(* CODESYS project Proyecto_Mezclador_de_alimenos_Codesys_V3_5_Sp12 (1).export

Project tree, tasks and I/O mapping:
  Device : CPX-CEC-C1-V3, Festo AG & Co. KG, order no. 3473128, version 3.5.12.60
      unmapped channels: Rotary switch
    application Application
      libraries: Standard, * (System); Util, * (System)
      task MainTask (cyclic, interval t#250MS, priority 20) calls LUCES, MODOMANUAL, CriaTilapia, TilapiaJoven, Tilapiaenengorda, GRANOSANIM, FlechasANIM, FORMULAS_Y_LLENADO_DE_SILOS, Alertas_silo, Alertas_SiloX
      global variables GVL
      image pool ImagePool
      image pool ImagePool_1
      program Alertas_silo [ST]
      program Alertas_SiloX [LD]
      program CriaTilapia [LD]
      program FlechasANIM [LD]
      program FORMULAS_Y_LLENADO_DE_SILOS [LD]
      program GRANOSANIM [LD]
      program LUCES [ST]
      program MODOMANUAL [LD]
      program Tilapiaenengorda [LD]
      program TilapiaJoven [LD]
      Symbols
      text list TextList
      visualisation Visualization
    PLC_Diagnosis : PLC-Diagnosis, Festo AG & Co. KG, version 3.5.4.3
    CPX_System : CPX_System, Festo AG & Co. KG, order no. 3473128, version 1.278
*)

// Device/Application/GVL
VAR_GLOBAL
	
	ON: BOOL;
	OFF: BOOL;
	ResetS: BOOL;
	OPCIONES:INT;
	
	A1:REAL;
	A2:REAL;
	A3:REAL;
	
	VMotor1: REAL;
	VMotor2: REAL;
	VMotor3: REAL; 
	INICIO2: BOOL;
	
	SiloF: REAL;
	LSiloF: BOOL;
	
	APAGADO: BOOL;
	Apagado2: BOOL;
	
	LMotor1: BOOL;
	LMotor2: BOOL;
	LMotor3: BOOL;
	
	
	MS: REAL;
	MTS1: REAL;
	MTS2: REAL;
	MTS3: REAL;
	PF1: REAL;
	PF2: REAL;
	PF3: REAL;
	
	Msn1: STRING;
	Msn2: STRING;
	Msn3: STRING;
	Msn4: STRING;
	
	OcultarB:BOOL;
	
	G1: BOOL;
	G3: BOOL;
	
	
	VaciadoF:BOOL;
	
	Luz1: BOOL;
	Luz2: BOOL;
	Luz3: BOOL;
	
	MSN5: STRING;
	MSN6: STRING;
	MSN7: STRING;
	
	img1: BOOL;
	img2: BOOL;
	img3: BOOL;
	
END_VAR

// Device/Application/LUCES
PROGRAM LUCES
VAR
END_VAR

/// Asignacion de variables para luces de silos
IF VMotor1 > 1 THEN;
	LMotor1:= TRUE ;
	ELSE
		LMotor1:= FALSE;
	END_IF
IF VMotor2 > 1 THEN;
	LMotor2:= TRUE ;
	ELSE
		LMotor2:= FALSE;
	END_IF
IF VMotor3 > 1 THEN;
	LMotor3:= TRUE ;
	ELSE
		LMotor3:= FALSE;
	END_IF

END_PROGRAM

// Device/Application/MODOMANUAL
PROGRAM MODOMANUAL
VAR
	G5: BOOL;
	Limite: BOOL;
	
END_VAR
VAR // added by the converter: edge detectors and wires of the graphical bodies
    _w1, _w2, _w3, _w4, _w5 : BOOL;
END_VAR

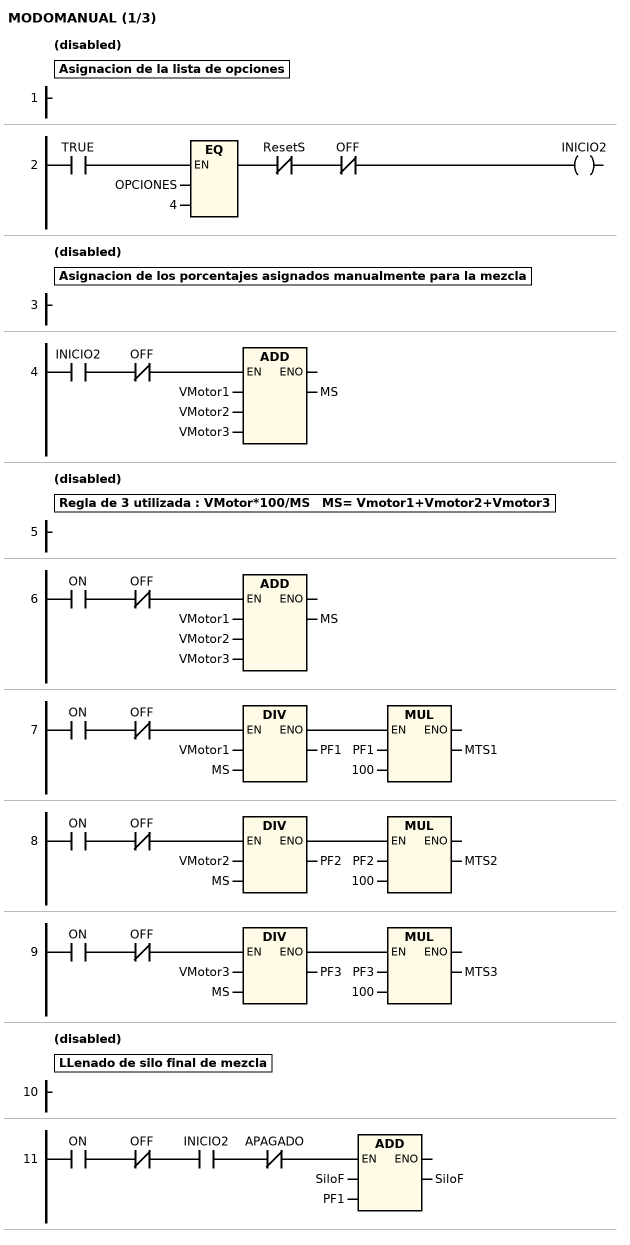
// NETWORK 1 (disabled)
// label: Asignacion de la lista de opciones

// NETWORK 2
INICIO2 := OPCIONES = 4 AND NOT ResetS AND NOT OFF;

// NETWORK 3 (disabled)
// label: Asignacion de los porcentajes asignados manualmente para la mezcla

// NETWORK 4
IF INICIO2 AND NOT OFF THEN MS := VMotor1 + VMotor2 + VMotor3; END_IF

// NETWORK 5 (disabled)
// label: Regla de 3 utilizada : VMotor*100/MS   MS= Vmotor1+Vmotor2+Vmotor3

// NETWORK 6
IF ON AND NOT OFF THEN MS := VMotor1 + VMotor2 + VMotor3; END_IF

// NETWORK 7
_w1 := ON AND NOT OFF;
IF _w1 THEN PF1 := VMotor1 / MS; END_IF
IF _w1 THEN MTS1 := PF1 * 100; END_IF

// NETWORK 8
_w2 := ON AND NOT OFF;
IF _w2 THEN PF2 := VMotor2 / MS; END_IF
IF _w2 THEN MTS2 := PF2 * 100; END_IF

// NETWORK 9
_w3 := ON AND NOT OFF;
IF _w3 THEN PF3 := VMotor3 / MS; END_IF
IF _w3 THEN MTS3 := PF3 * 100; END_IF

// NETWORK 10 (disabled)
// label: LLenado de silo final de mezcla

// NETWORK 11
IF ON AND NOT OFF AND INICIO2 AND NOT APAGADO THEN SiloF := SiloF + PF1; END_IF

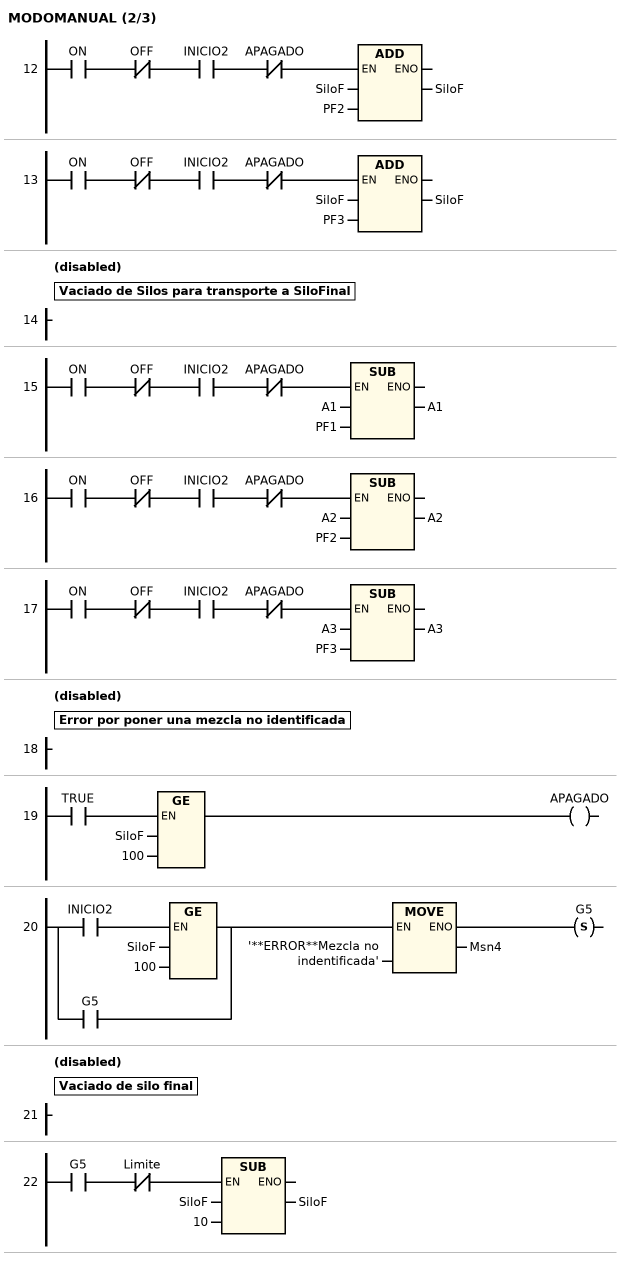
// NETWORK 12
IF ON AND NOT OFF AND INICIO2 AND NOT APAGADO THEN SiloF := SiloF + PF2; END_IF

// NETWORK 13
IF ON AND NOT OFF AND INICIO2 AND NOT APAGADO THEN SiloF := SiloF + PF3; END_IF

// NETWORK 14 (disabled)
// label: Vaciado de Silos para transporte a SiloFinal

// NETWORK 15
IF ON AND NOT OFF AND INICIO2 AND NOT APAGADO THEN A1 := A1 - PF1; END_IF

// NETWORK 16
IF ON AND NOT OFF AND INICIO2 AND NOT APAGADO THEN A2 := A2 - PF2; END_IF

// NETWORK 17
IF ON AND NOT OFF AND INICIO2 AND NOT APAGADO THEN A3 := A3 - PF3; END_IF

// NETWORK 18 (disabled)
// label: Error por poner una mezcla no identificada

// NETWORK 19
APAGADO := SiloF >= 100;

// NETWORK 20
_w4 := INICIO2 AND SiloF >= 100 OR G5;
IF _w4 THEN Msn4 := '**ERROR**Mezcla no indentificada'; END_IF
G5 S= _w4;

// NETWORK 21 (disabled)
// label: Vaciado de silo final

// NETWORK 22
IF G5 AND NOT Limite THEN SiloF := SiloF - 10; END_IF

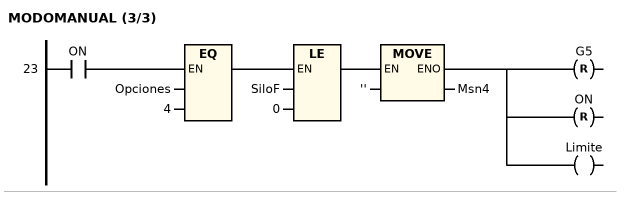
// NETWORK 23
_w5 := ON AND Opciones = 4 AND SiloF <= 0;
IF _w5 THEN Msn4 := ''; END_IF
G5 R= _w5;
ON R= _w5;
Limite := _w5;

END_PROGRAM

// Device/Application/CriaTilapia
PROGRAM CriaTilapia
VAR
	INICIO1: BOOL;
	ENCENDIDO1: BOOL;
	CERO1: BOOL;
	CERO2: BOOL;
	CERO3: BOOL;
	imagen1: BOOL;
	
END_VAR
VAR // added by the converter: edge detectors and wires of the graphical bodies
    _w1, _w2, _w3 : BOOL;
END_VAR

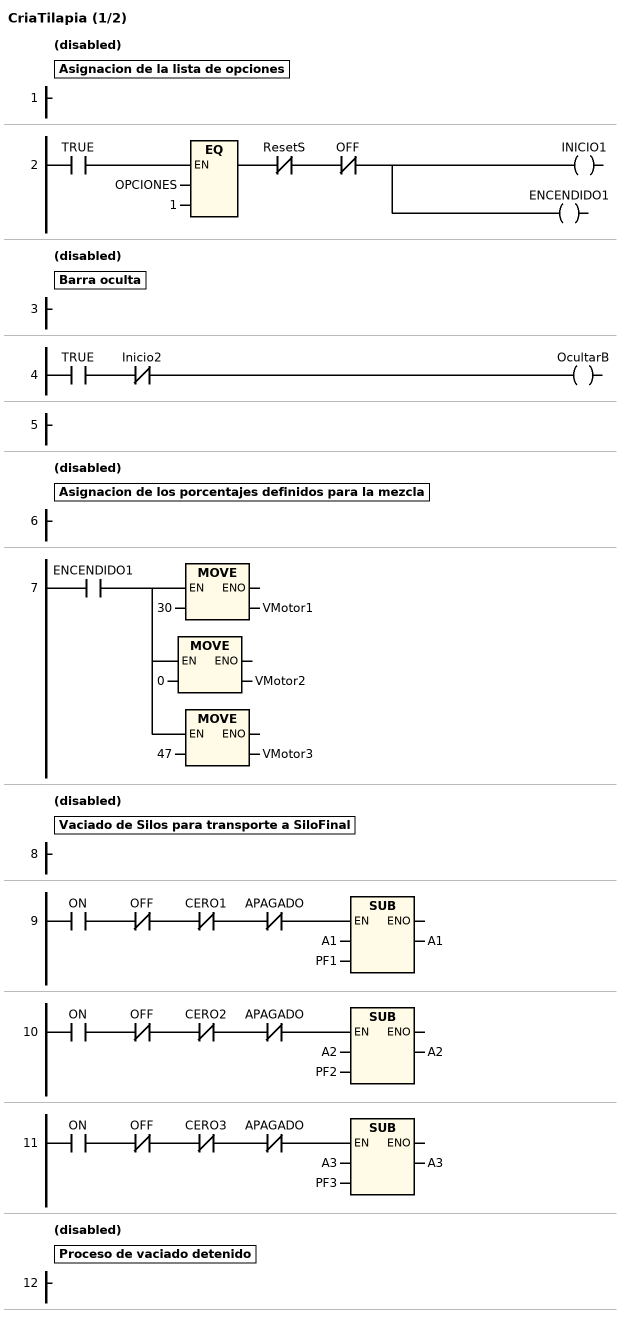
// NETWORK 1 (disabled)
// label: Asignacion de la lista de opciones

// NETWORK 2
_w1 := OPCIONES = 1 AND NOT ResetS AND NOT OFF;
INICIO1 := _w1;
ENCENDIDO1 := _w1;

// NETWORK 3 (disabled)
// label: Barra oculta

// NETWORK 4
OcultarB := TRUE AND NOT Inicio2;

// NETWORK 5

// NETWORK 6 (disabled)
// label: Asignacion de los porcentajes definidos para la mezcla

// NETWORK 7
IF ENCENDIDO1 THEN VMotor1 := 30; END_IF
IF ENCENDIDO1 THEN VMotor2 := 0; END_IF
IF ENCENDIDO1 THEN VMotor3 := 47; END_IF

// NETWORK 8 (disabled)
// label: Vaciado de Silos para transporte a SiloFinal

// NETWORK 9
IF ON AND NOT OFF AND NOT CERO1 AND NOT APAGADO THEN A1 := A1 - PF1; END_IF

// NETWORK 10
IF ON AND NOT OFF AND NOT CERO2 AND NOT APAGADO THEN A2 := A2 - PF2; END_IF

// NETWORK 11
IF ON AND NOT OFF AND NOT CERO3 AND NOT APAGADO THEN A3 := A3 - PF3; END_IF

// NETWORK 12 (disabled)
// label: Proceso de vaciado detenido

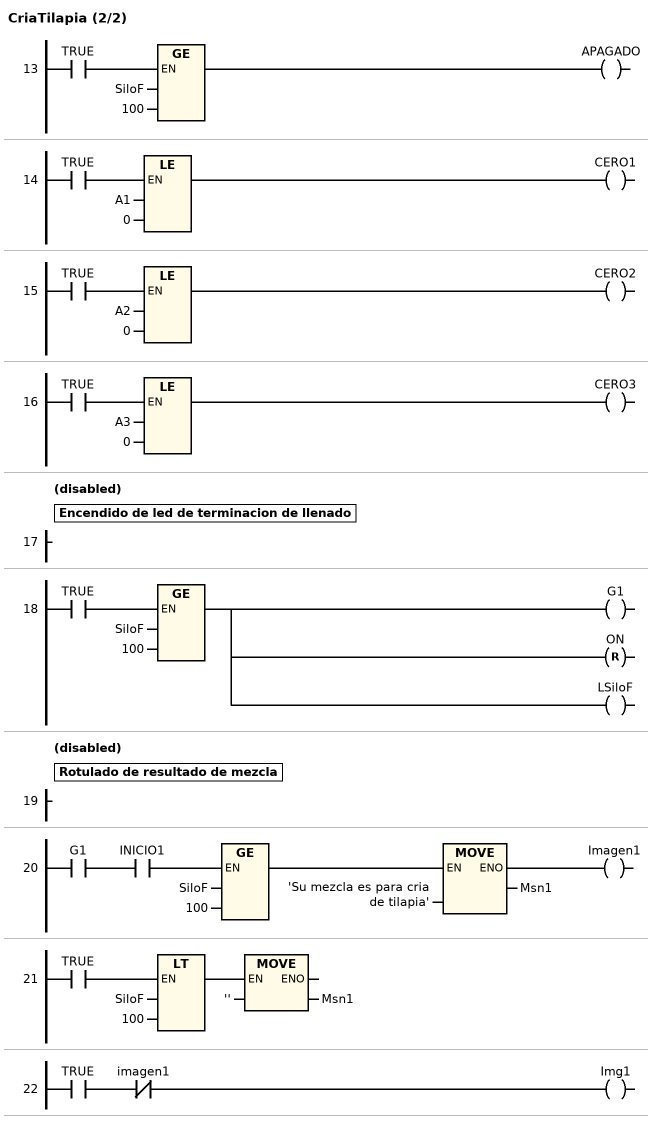
// NETWORK 13
APAGADO := SiloF >= 100;

// NETWORK 14
CERO1 := A1 <= 0;

// NETWORK 15
CERO2 := A2 <= 0;

// NETWORK 16
CERO3 := A3 <= 0;

// NETWORK 17 (disabled)
// label: Encendido de led de terminacion de llenado

// NETWORK 18
_w2 := SiloF >= 100;
G1 := _w2;
ON R= _w2;
LSiloF := _w2;

// NETWORK 19 (disabled)
// label: Rotulado de resultado de mezcla

// NETWORK 20
_w3 := G1 AND INICIO1 AND SiloF >= 100;
IF _w3 THEN Msn1 := 'Su mezcla es para cria de tilapia'; END_IF
Imagen1 := _w3;

// NETWORK 21
IF SiloF < 100 THEN Msn1 := ''; END_IF

// NETWORK 22
Img1 := TRUE AND NOT imagen1;

END_PROGRAM

// Device/Application/TilapiaJoven
PROGRAM TilapiaJoven
VAR
	INICIO3: BOOL;
	ENCENDIDO2: BOOL;
	CERO4: BOOL;
	CERO5: BOOL;
	CERO6: BOOL;
	G2: BOOL;
	imagen2: BOOL;
END_VAR
VAR // added by the converter: edge detectors and wires of the graphical bodies
    _w1, _w2, _w3 : BOOL;
END_VAR

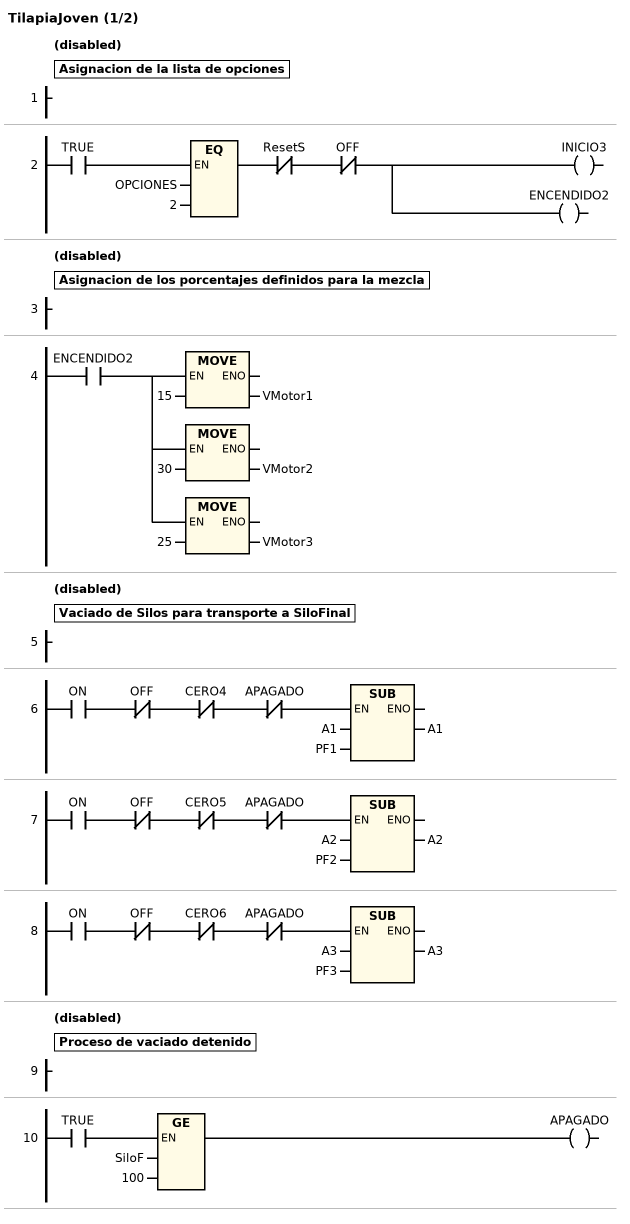
// NETWORK 1 (disabled)
// label: Asignacion de la lista de opciones

// NETWORK 2
_w1 := OPCIONES = 2 AND NOT ResetS AND NOT OFF;
INICIO3 := _w1;
ENCENDIDO2 := _w1;

// NETWORK 3 (disabled)
// label: Asignacion de los porcentajes definidos para la mezcla

// NETWORK 4
IF ENCENDIDO2 THEN VMotor1 := 15; END_IF
IF ENCENDIDO2 THEN VMotor2 := 30; END_IF
IF ENCENDIDO2 THEN VMotor3 := 25; END_IF

// NETWORK 5 (disabled)
// label: Vaciado de Silos para transporte a SiloFinal

// NETWORK 6
IF ON AND NOT OFF AND NOT CERO4 AND NOT APAGADO THEN A1 := A1 - PF1; END_IF

// NETWORK 7
IF ON AND NOT OFF AND NOT CERO5 AND NOT APAGADO THEN A2 := A2 - PF2; END_IF

// NETWORK 8
IF ON AND NOT OFF AND NOT CERO6 AND NOT APAGADO THEN A3 := A3 - PF3; END_IF

// NETWORK 9 (disabled)
// label: Proceso de vaciado detenido

// NETWORK 10
APAGADO := SiloF >= 100;

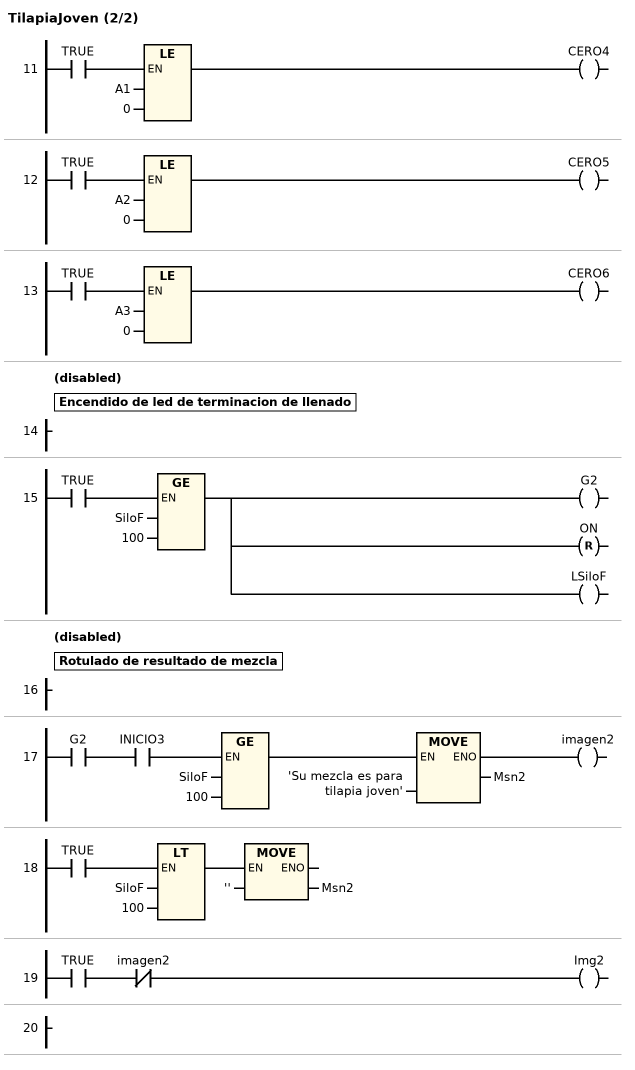
// NETWORK 11
CERO4 := A1 <= 0;

// NETWORK 12
CERO5 := A2 <= 0;

// NETWORK 13
CERO6 := A3 <= 0;

// NETWORK 14 (disabled)
// label: Encendido de led de terminacion de llenado

// NETWORK 15
_w2 := SiloF >= 100;
G2 := _w2;
ON R= _w2;
LSiloF := _w2;

// NETWORK 16 (disabled)
// label: Rotulado de resultado de mezcla

// NETWORK 17
_w3 := G2 AND INICIO3 AND SiloF >= 100;
IF _w3 THEN Msn2 := 'Su mezcla es para tilapia joven'; END_IF
imagen2 := _w3;

// NETWORK 18
IF SiloF < 100 THEN Msn2 := ''; END_IF

// NETWORK 19
Img2 := TRUE AND NOT imagen2;

// NETWORK 20

END_PROGRAM

// Device/Application/Tilapiaenengorda
PROGRAM Tilapiaenengorda
VAR
	INICIO4: BOOL;
	ENCENDIDO3: BOOL;
	CERO7: BOOL;
	CERO8: BOOL;
	CERO9: BOOL;
	
	
	imagen2: BOOL;
END_VAR
VAR // added by the converter: edge detectors and wires of the graphical bodies
    _w1, _w2, _w3 : BOOL;
END_VAR

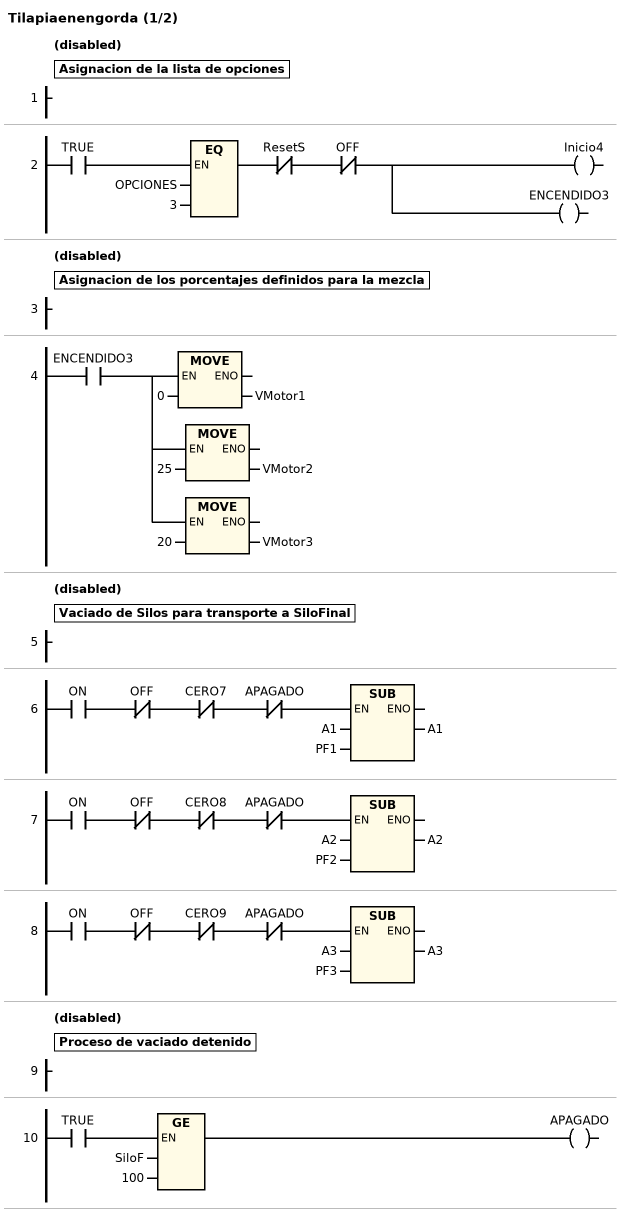
// NETWORK 1 (disabled)
// label: Asignacion de la lista de opciones

// NETWORK 2
_w1 := OPCIONES = 3 AND NOT ResetS AND NOT OFF;
Inicio4 := _w1;
ENCENDIDO3 := _w1;

// NETWORK 3 (disabled)
// label: Asignacion de los porcentajes definidos para la mezcla

// NETWORK 4
IF ENCENDIDO3 THEN VMotor1 := 0; END_IF
IF ENCENDIDO3 THEN VMotor2 := 25; END_IF
IF ENCENDIDO3 THEN VMotor3 := 20; END_IF

// NETWORK 5 (disabled)
// label: Vaciado de Silos para transporte a SiloFinal

// NETWORK 6
IF ON AND NOT OFF AND NOT CERO7 AND NOT APAGADO THEN A1 := A1 - PF1; END_IF

// NETWORK 7
IF ON AND NOT OFF AND NOT CERO8 AND NOT APAGADO THEN A2 := A2 - PF2; END_IF

// NETWORK 8
IF ON AND NOT OFF AND NOT CERO9 AND NOT APAGADO THEN A3 := A3 - PF3; END_IF

// NETWORK 9 (disabled)
// label: Proceso de vaciado detenido

// NETWORK 10
APAGADO := SiloF >= 100;

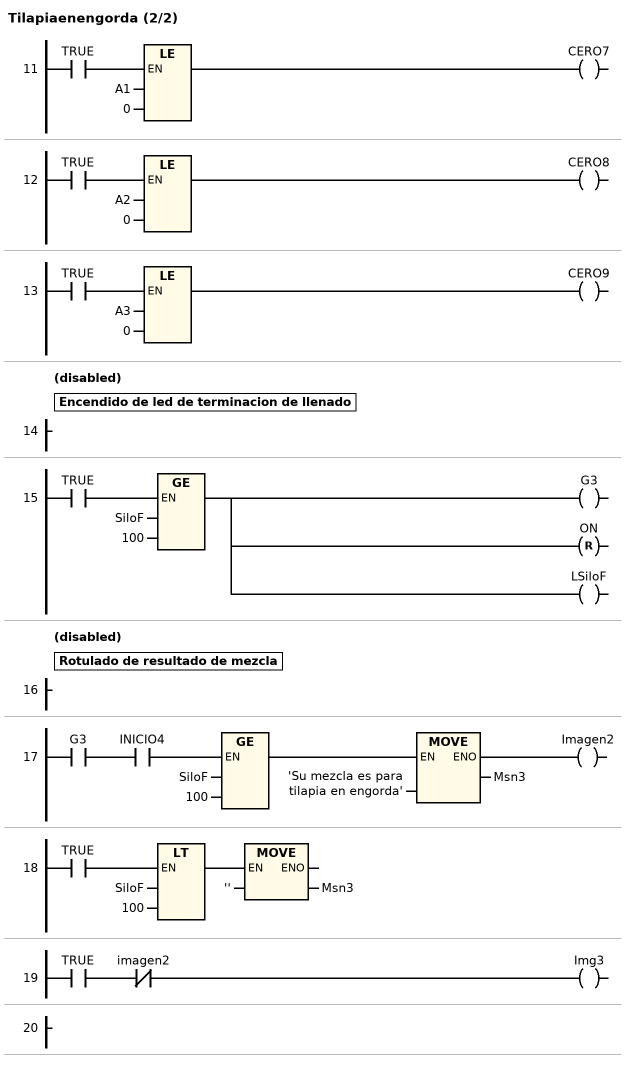
// NETWORK 11
CERO7 := A1 <= 0;

// NETWORK 12
CERO8 := A2 <= 0;

// NETWORK 13
CERO9 := A3 <= 0;

// NETWORK 14 (disabled)
// label: Encendido de led de terminacion de llenado

// NETWORK 15
_w2 := SiloF >= 100;
G3 := _w2;
ON R= _w2;
LSiloF := _w2;

// NETWORK 16 (disabled)
// label: Rotulado de resultado de mezcla

// NETWORK 17
_w3 := G3 AND INICIO4 AND SiloF >= 100;
IF _w3 THEN Msn3 := 'Su mezcla es para tilapia en engorda'; END_IF
Imagen2 := _w3;

// NETWORK 18
IF SiloF < 100 THEN Msn3 := ''; END_IF

// NETWORK 19
Img3 := TRUE AND NOT imagen2;

// NETWORK 20

END_PROGRAM

// Device/Application/GRANOSANIM
PROGRAM GRANOSANIM
VAR
	IPOSY: INT;
	Blink1: BLINK;
	MOV1: BOOL;
	R_TRIG_1: R_TRIG;
	MOV2: BOOL;
	STOP2: BOOL;
	R_TRIG_2: R_TRIG;
END_VAR
VAR // added by the converter: edge detectors and wires of the graphical bodies
    _w1 : BOOL;
END_VAR

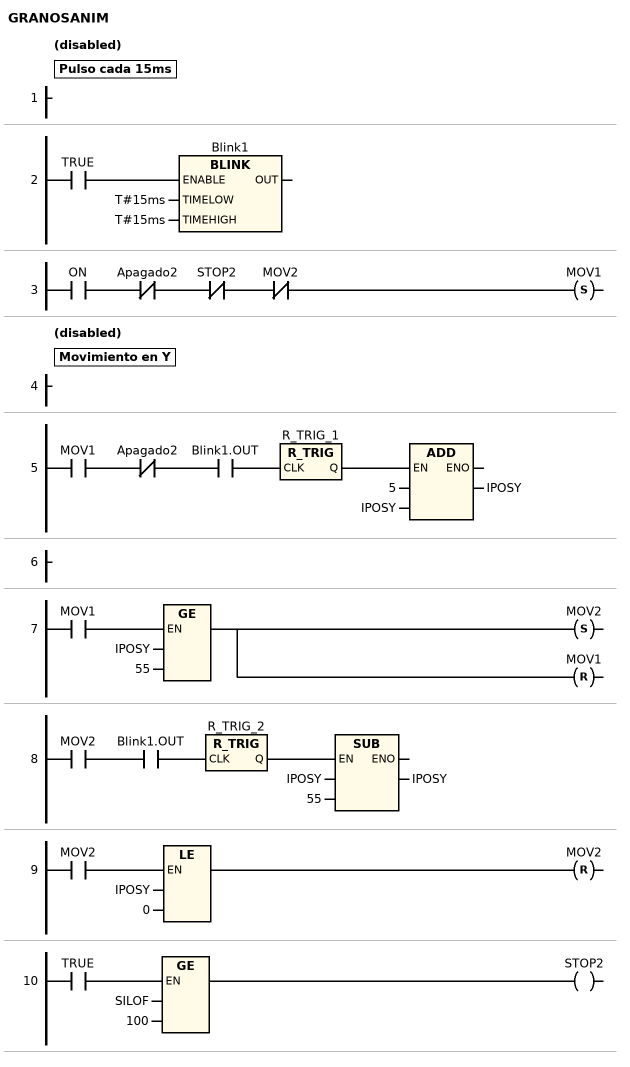
// NETWORK 1 (disabled)
// label: Pulso cada 15ms

// NETWORK 2
Blink1(ENABLE := TRUE, TIMELOW := T#15ms, TIMEHIGH := T#15ms); // BLINK

// NETWORK 3
MOV1 S= ON AND NOT Apagado2 AND NOT STOP2 AND NOT MOV2;

// NETWORK 4 (disabled)
// label: Movimiento en Y

// NETWORK 5
R_TRIG_1(CLK := MOV1 AND NOT Apagado2 AND Blink1.OUT); // R_TRIG
IF R_TRIG_1.Q THEN IPOSY := 5 + IPOSY; END_IF

// NETWORK 6

// NETWORK 7
_w1 := MOV1 AND IPOSY >= 55;
MOV2 S= _w1;
MOV1 R= _w1;

// NETWORK 8
R_TRIG_2(CLK := MOV2 AND Blink1.OUT); // R_TRIG
IF R_TRIG_2.Q THEN IPOSY := IPOSY - 55; END_IF

// NETWORK 9
MOV2 R= MOV2 AND IPOSY <= 0;

// NETWORK 10
STOP2 := SILOF >= 100;

END_PROGRAM

// Device/Application/FlechasANIM
PROGRAM FlechasANIM
VAR
	Blink2: BLINK;
	STOP3: BOOL;
	MOV3: BOOL;
	R_TRIG_4: R_TRIG;
	R_TRIG_3: R_TRIG;
	IPOSX:INT;
	MOV4: BOOL;
END_VAR
VAR // added by the converter: edge detectors and wires of the graphical bodies
    _w1 : BOOL;
END_VAR

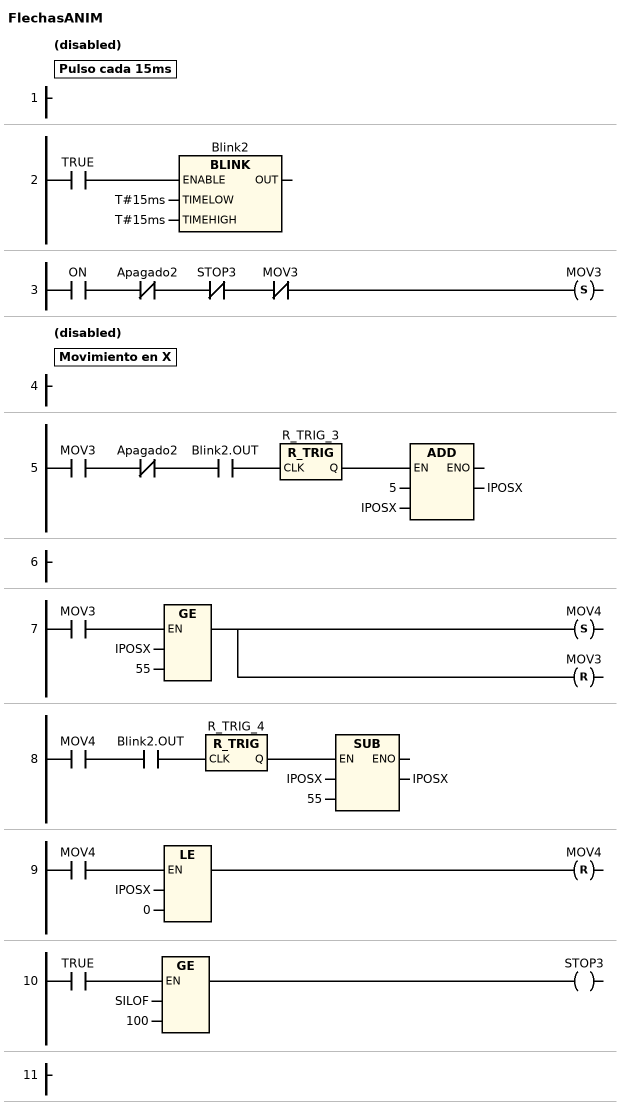
// NETWORK 1 (disabled)
// label: Pulso cada 15ms

// NETWORK 2
Blink2(ENABLE := TRUE, TIMELOW := T#15ms, TIMEHIGH := T#15ms); // BLINK

// NETWORK 3
MOV3 S= ON AND NOT Apagado2 AND NOT STOP3 AND NOT MOV3;

// NETWORK 4 (disabled)
// label: Movimiento en X

// NETWORK 5
R_TRIG_3(CLK := MOV3 AND NOT Apagado2 AND Blink2.OUT); // R_TRIG
IF R_TRIG_3.Q THEN IPOSX := 5 + IPOSX; END_IF

// NETWORK 6

// NETWORK 7
_w1 := MOV3 AND IPOSX >= 55;
MOV4 S= _w1;
MOV3 R= _w1;

// NETWORK 8
R_TRIG_4(CLK := MOV4 AND Blink2.OUT); // R_TRIG
IF R_TRIG_4.Q THEN IPOSX := IPOSX - 55; END_IF

// NETWORK 9
MOV4 R= MOV4 AND IPOSX <= 0;

// NETWORK 10
STOP3 := SILOF >= 100;

// NETWORK 11

END_PROGRAM

// Device/Application/FORMULAS_Y_LLENADO_DE_SILOS
PROGRAM FORMULAS_Y_LLENADO_DE_SILOS
VAR
	SiloFULL: BOOL;
	SiloLL: BOOL;
	B1: REAL;
	B2: REAL;
	B3: REAL;
	Limite1: BOOL;
	Ajuste: BOOL;
END_VAR
VAR // added by the converter: edge detectors and wires of the graphical bodies
    _w1, _w2, _w3, _w4, _w5, _w6, _w7, _w8 : BOOL;
END_VAR

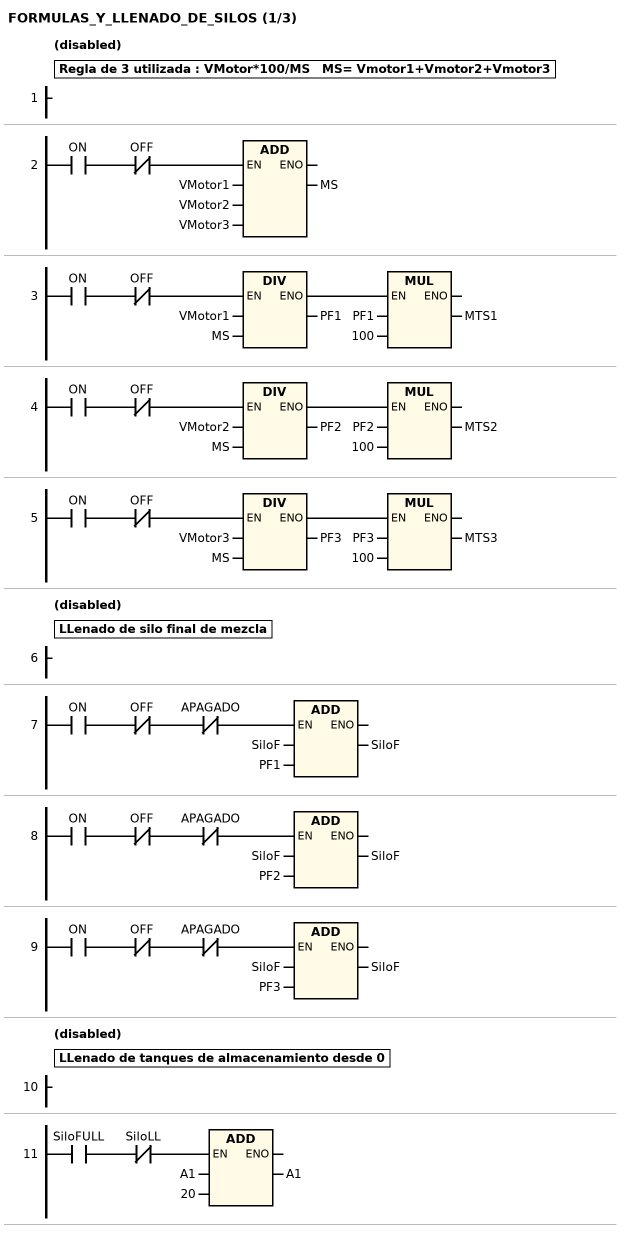
// NETWORK 1 (disabled)
// label: Regla de 3 utilizada : VMotor*100/MS   MS= Vmotor1+Vmotor2+Vmotor3

// NETWORK 2
IF ON AND NOT OFF THEN MS := VMotor1 + VMotor2 + VMotor3; END_IF

// NETWORK 3
_w1 := ON AND NOT OFF;
IF _w1 THEN PF1 := VMotor1 / MS; END_IF
IF _w1 THEN MTS1 := PF1 * 100; END_IF

// NETWORK 4
_w2 := ON AND NOT OFF;
IF _w2 THEN PF2 := VMotor2 / MS; END_IF
IF _w2 THEN MTS2 := PF2 * 100; END_IF

// NETWORK 5
_w3 := ON AND NOT OFF;
IF _w3 THEN PF3 := VMotor3 / MS; END_IF
IF _w3 THEN MTS3 := PF3 * 100; END_IF

// NETWORK 6 (disabled)
// label: LLenado de silo final de mezcla

// NETWORK 7
IF ON AND NOT OFF AND NOT APAGADO THEN SiloF := SiloF + PF1; END_IF

// NETWORK 8
IF ON AND NOT OFF AND NOT APAGADO THEN SiloF := SiloF + PF2; END_IF

// NETWORK 9
IF ON AND NOT OFF AND NOT APAGADO THEN SiloF := SiloF + PF3; END_IF

// NETWORK 10 (disabled)
// label: LLenado de tanques de almacenamiento desde 0

// NETWORK 11
IF SiloFULL AND NOT SiloLL THEN A1 := A1 + 20; END_IF

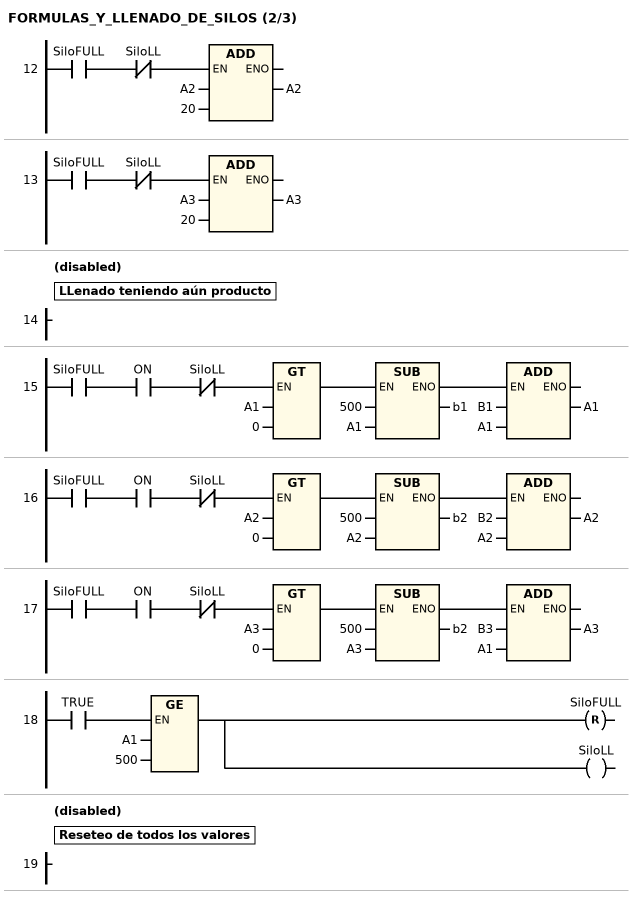
// NETWORK 12
IF SiloFULL AND NOT SiloLL THEN A2 := A2 + 20; END_IF

// NETWORK 13
IF SiloFULL AND NOT SiloLL THEN A3 := A3 + 20; END_IF

// NETWORK 14 (disabled)
// label: LLenado teniendo aún producto

// NETWORK 15
_w4 := SiloFULL AND ON AND NOT SiloLL AND A1 > 0;
IF _w4 THEN b1 := 500 - A1; END_IF
IF _w4 THEN A1 := B1 + A1; END_IF

// NETWORK 16
_w5 := SiloFULL AND ON AND NOT SiloLL AND A2 > 0;
IF _w5 THEN b2 := 500 - A2; END_IF
IF _w5 THEN A2 := B2 + A2; END_IF

// NETWORK 17
_w6 := SiloFULL AND ON AND NOT SiloLL AND A3 > 0;
IF _w6 THEN b2 := 500 - A3; END_IF
IF _w6 THEN A3 := B3 + A1; END_IF

// NETWORK 18
_w7 := A1 >= 500;
SiloFULL R= _w7;
SiloLL := _w7;

// NETWORK 19 (disabled)
// label: Reseteo de todos los valores

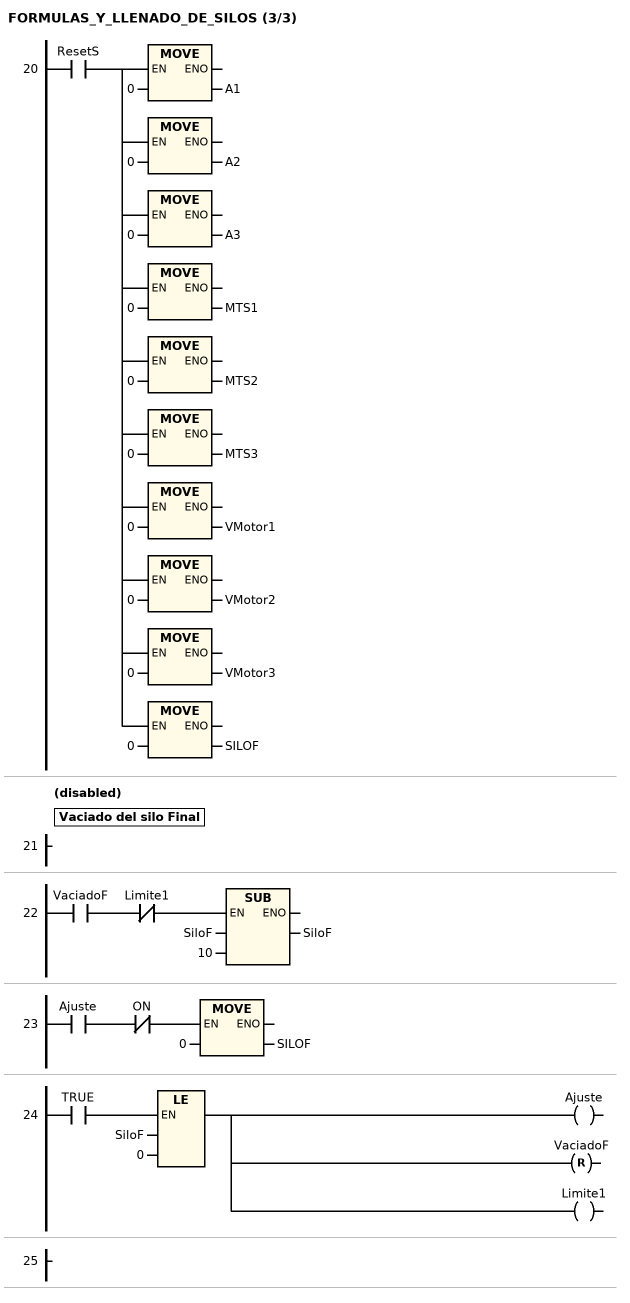
// NETWORK 20
IF ResetS THEN A1 := 0; END_IF
IF ResetS THEN A2 := 0; END_IF
IF ResetS THEN A3 := 0; END_IF
IF ResetS THEN MTS1 := 0; END_IF
IF ResetS THEN MTS2 := 0; END_IF
IF ResetS THEN MTS3 := 0; END_IF
IF ResetS THEN VMotor1 := 0; END_IF
IF ResetS THEN VMotor2 := 0; END_IF
IF ResetS THEN VMotor3 := 0; END_IF
IF ResetS THEN SILOF := 0; END_IF

// NETWORK 21 (disabled)
// label: Vaciado del silo Final

// NETWORK 22
IF VaciadoF AND NOT Limite1 THEN SiloF := SiloF - 10; END_IF

// NETWORK 23
IF Ajuste AND NOT ON THEN SILOF := 0; END_IF

// NETWORK 24
_w8 := SiloF <= 0;
Ajuste := _w8;
VaciadoF R= _w8;
Limite1 := _w8;

// NETWORK 25

END_PROGRAM

// Device/Application/Alertas_silo
PROGRAM Alertas_silo
VAR
END_VAR

IF A1<= 200 THEN
	Luz1:= TRUE;
	ELSE
		Luz1:= FALSE;
	
END_IF
IF A2<= 200 THEN
	Luz2:= TRUE;
	ELSE
		Luz2:= FALSE;
	
END_IF
IF A3<= 200 THEN
	Luz3:= TRUE;
	ELSE
		Luz3:= FALSE;
	
END_IF
IF A3<=0 THEN
	OFF:= TRUE;
	ELSE  
		OFF:= FALSE ;
	END_IF

IF A3<=0 THEN;
	OFF:= TRUE;
	ELSE  
		OFF:= FALSE ;
	
END_IF
IF A3<=0 THEN;
	OFF:= TRUE;
	ELSE  
		OFF:= FALSE ;
	
END_IF

END_PROGRAM

// Device/Application/Alertas_SiloX
PROGRAM Alertas_SiloX
VAR
END_VAR

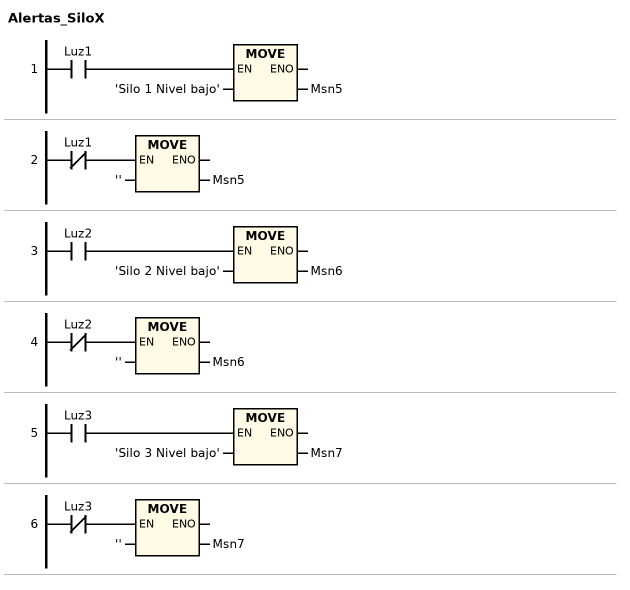
// NETWORK 1
IF Luz1 THEN Msn5 := 'Silo 1 Nivel bajo'; END_IF

// NETWORK 2
IF NOT Luz1 THEN Msn5 := ''; END_IF

// NETWORK 3
IF Luz2 THEN Msn6 := 'Silo 2 Nivel bajo'; END_IF

// NETWORK 4
IF NOT Luz2 THEN Msn6 := ''; END_IF

// NETWORK 5
IF Luz3 THEN Msn7 := 'Silo 3 Nivel bajo'; END_IF

// NETWORK 6
IF NOT Luz3 THEN Msn7 := ''; END_IF

END_PROGRAM

// Device/Application/Visualization
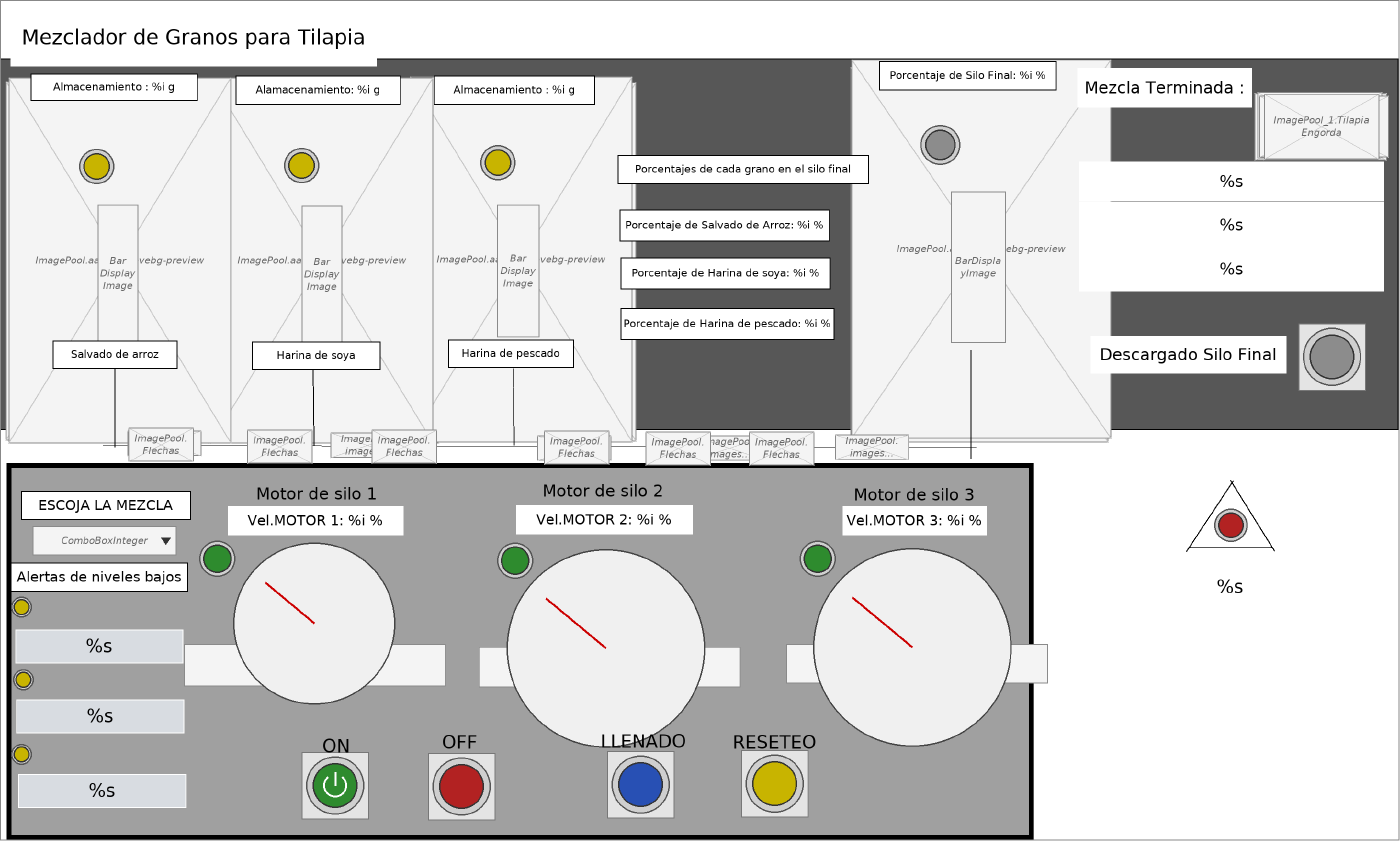
VISUALIZATION Visualization  // 1462x879
    RoundedRectangle (7,484 1072x393)
    RoundedRectangle (0,61 1460x388)
    Image (888,70 269x392), image: ImagePool.Diseños de Silo
    Image (424,86 240x375), image: ImagePool.Diseños de Silo
    Image (218,88 240x375), image: ImagePool.Diseños de Silo
    Image (6,85 240x375), image: ImagePool.Diseños de Silo
    Image (889,62 271x396), image: ImagePool.aaaa-removebg-preview
    Image (428,80 232x382), image: ImagePool.aaaa-removebg-preview
    Image (220,81 232x382), image: ImagePool.aaaa-removebg-preview
    Image (9,81 232x382), image: ImagePool.aaaa-removebg-preview
    Slider (821,673 273x41), variable: VMotor3, invisible if: OcultarB, scale 0..100
    Slider (500,676 273x42), variable: VMotor2, invisible if: OcultarB, scale 0..100
    Slider (192,673 273x44), variable: VMotor1, invisible if: OcultarB, scale 0..100
    Label (256,501 150x30), "Motor de silo 1"
    Label (555,498 150x30), "Motor de silo 2"
    Label (880,502 150x30), "Motor de silo 3"
    Line (120,467) (120,385)
    Line (328,465) (327,383)
    Line (537,465) (536,385)
    Line (108,465) (1019,467)
    Line (1014,479) (1014,366)
    BarDisplayImage (993,200 57x158), value: SiloF, style: BarDisplayImage-Gray, scale format: %.1f, scale 0..100
    Meter180 (226,567 204x169), value: VMotor1, style: Meter-Meter180-Yellow, scale format: %.1f, scale 0..100
        p518627256: %
    Meter180 (529,565 207x225), value: VMotor2, style: Meter-Meter180-Yellow, scale format: %.1f, scale 0..100
        p518627256: %
    Meter180 (849,564 207x225), value: VMotor3, style: Meter-Meter180-Yellow, scale format: %.1f, scale 0..100
        p518627256: %
    Lamp1 (512,564 52x44), variable: LMotor2, style: Lamp-Lamp1-Green
    Lamp1 (201,562 52x44), variable: LMotor1, style: Lamp-Lamp1-Green
    Lamp1 (828,562 52x44), variable: LMotor3, style: Lamp-Lamp1-Green
    RoundedRectangle (453,79 168x30), "Almacenamiento : %i g", text variable: A3
    RoundedRectangle (246,79 172x30), "Alamacenamiento: %i g", text variable: A2
    RoundedRectangle (32,77 174x28), "Almacenamiento : %i g", text variable: A1
    RoundedRectangle (918,64 185x30), "Porcentaje de Silo Final: %i %", text variable: SiloF
    PowerSwitch (315,786 70x70), variable: ON, behaviour: TOGGLE, style: Switch-PowerSwitch-Green
    PushSwitch (447,787 70x70), variable: OFF, behaviour: TOGGLE, style: Switch-PushSwitch-Red
    Lamp1 (958,125 48x53), variable: LSiloF, style: Lamp-Lamp1-Gray
    BarDisplayImage (102,214 42x143), value: A1, style: BarDisplayImage-Gray, scale format: %.1f, scale 0..500
    BarDisplayImage (315,215 42x143), value: A2, style: BarDisplayImage-Gray, scale format: %.1f, scale 0..500
    BarDisplayImage (519,214 44x138), value: A3, style: BarDisplayImage-Gray, scale format: %.1f, scale 0..500
    Label (276,765 150x30), "ON"
    RoundedRectangle (880,529 150x30), "Vel.MOTOR 3: %i %", text variable: VMotor3
    RoundedRectangle (539,528 184x30), "Vel.MOTOR 2: %i %", text variable: VMotor2
    RoundedRectangle (238,529 183x30), "Vel.MOTOR 1: %i %", text variable: VMotor1
    Label (405,761 150x30), "OFF"
    RoundedRectangle (647,219 219x33), "Porcentaje de Salvado de Arroz: %i %", text variable: MTS1
    RoundedRectangle (648,269 219x33), "Porcentaje de Harina de soya: %i %", text variable: MTS2
    RoundedRectangle (648,322 223x33), "Porcentaje de Harina de pescado: %i %", text variable: MTS3
    PushSwitch (634,785 70x70), variable: FORMULAS_Y_LLENADO_DE_SILOS.SiloFULL, behaviour: TOGGLE, style: Switch-PushSwitch-Blue
    PushSwitch (774,784 70x70), variable: ResetS, behaviour: TOGGLE, style: Switch-PushSwitch-Yellow
    ComboBoxInteger (34,550 150x30), variable: OPCIONES, text list: 'TextList'
        p1601986498: ''
    RoundedRectangle (22,513 177x30), "ESCOJA LA MEZCLA"
    Label (734,761 150x30), "RESETEO"
    Label (597,760 150x30), "LLENADO"
    Rectangle (1127,169 318x41), "%s", text variable: Msn1
    Rectangle (1125,71 182x41), "Mezcla Terminada :"
    Rectangle (1127,211 318x48), "%s", text variable: MSN2
    Rectangle (1127,258 318x46), "%s", text variable: Msn3
    RoundedRectangle (11,9 382x60), "Mezclador de Granos para Tilapia"
    Rectangle (55,356 130x29), "Salvado de arroz"
    Rectangle (263,357 134x29), "Harina de soya"
    Rectangle (468,355 131x29), "Harina de pescado"
    PushSwitch (1356,338 70x70), variable: VaciadoF, behaviour: TOGGLE, style: Switch-PushSwitch-Gray
    Rectangle (1139,351 204x39), "Descargado Silo Final"
    Image (133,450 77x26), image: ImagePool.images-removebg-preview
        p3560616238: FlechasANIM.IPOSX
    Image (345,452 77x26), image: ImagePool.images-removebg-preview
        p3560616238: FlechasANIM.IPOSX
    Image (561,455 77x26), image: ImagePool.images-removebg-preview
        p3560616238: FlechasANIM.IPOSX
    Image (723,455 77x26), image: ImagePool.images-removebg-preview
        p3560616238: FlechasANIM.IPOSX
    Image (872,454 77x26), image: ImagePool.images-removebg-preview
        p3560616238: FlechasANIM.IPOSX
    Line (1239,576) (1288,502)
    Line (1331,576) (1285,502)
    Line (1241,572) (1329,572)
    Lamp1 (1265,529 41x40), variable: MODOMANUAL.G5, style: Lamp-Lamp1-Red
    Rectangle (1120,585 329x57), "%s", text variable: Msn4
    RoundedRectangle (645,162 262x30), "Porcentajes de cada grano en el silo final"
    Lamp1 (80,151 42x46), variable: Luz1, style: Lamp-Lamp1-Yellow
    Lamp1 (294,150 42x46), variable: Luz2, style: Lamp-Lamp1-Yellow
    Lamp1 (499,147 42x46), variable: Luz3, style: Lamp-Lamp1-Yellow
    Lamp1 (10,622 25x25), variable: Luz1, style: Lamp-Lamp1-Yellow
    Rectangle (16,658 175x35), "%s", text variable: MSN6
    Lamp1 (10,776 25x25), variable: Luz3, style: Lamp-Lamp1-Yellow
    Lamp1 (12,698 25x25), variable: Luz2, style: Lamp-Lamp1-Yellow
    Rectangle (17,731 175x35), "%s", text variable: MSN5
    Rectangle (19,809 175x35), "%s", text variable: MSN7
    RoundedRectangle (11,588 185x30), "Alertas de niveles bajos"
    Image (1319,104 128x63), invisible if: img1, image: ImagePool_1.5ceeeef3a84b7e0015bd153c-ZGL31005-1
    Image (1310,97 138x70), invisible if: img2, image: ImagePool_1.Oreo_nilo_071011-0507_F_jtg
    Image (1314,101 129x63), invisible if: img3, image: ImagePool_1.Tilapia_Azul
    Image (1313,96 130x69), invisible if: img1, image: ImagePool_1.Cria deTilapia
    Image (1315,100 135x64), invisible if: img2, image: ImagePool_1.Tilapia Juvenil
    Image (1320,98 120x68), invisible if: img3, image: ImagePool_1.Tilapia Engorda
    Image (134,447 68x35), image: ImagePool.Flechas
        p3560616238: FlechasANIM.IPOSX
    Image (258,449 68x35), image: ImagePool.Flechas
        p3560616238: FlechasANIM.IPOSX
    Image (388,449 68x35), image: ImagePool.Flechas
        p3560616238: FlechasANIM.IPOSX
    Image (568,450 68x35), image: ImagePool.Flechas
        p3560616238: FlechasANIM.IPOSX
    Image (674,451 68x35), image: ImagePool.Flechas
        p3560616238: FlechasANIM.IPOSX
    Image (782,451 68x35), image: ImagePool.Flechas
        p3560616238: FlechasANIM.IPOSX
END_VISUALIZATION

(* text list TextList (id | default)
  1 | Cria de tilapia
  2 | Tilapia Joven
  3 | Tilapia en engorda
  4 | MANUAL
   |  *)
